// TIA Portal V17 export
// export: Created 2023-12-22T15:03:03.5721321Z, ExportSetting WithDefaults, DisplayName Totally Integrated Automation Portal, DisplayVersion V17, DisplayName TIA Portal Openness, DisplayVersion V17, DisplayName TIA Portal Version Control Interface, DisplayVersion V17, DisplayName STEP 7 Professional, DisplayVersion V17, DisplayName STEP 7 Safety, DisplayVersion V17, DisplayName WinCC Advanced, DisplayVersion V17
DATA_BLOCK "PIDx_DB"   // DB260
VERSION : 0.1
// stored: AutoNumber false, DBAccessibleFromOPCUA true, DBAccessibleFromWebserver true, InstanceOfName PIDx, InstanceOfType FB
"PIDx"
   // VAR RETAIN
   //    Time_DTL { S7_SetPoint := 'True'} : DTL := DTL#2023-05-02-18:36:48.871840937;
   // END_VAR
BEGIN
END_DATA_BLOCK
